PROGRAM MAIN
VAR
	iCounter 	: INT;
	
	bToggle		: BOOL;
	bReset		: BOOL;
	sText		: STRING; 
	
	stMyVar		: ST_MyType;
END_VAR


IF bToggle THEN
	sText := 'Stop';
	iCounter := (iCounter + 1) MOD 1000;
	IF iCounter = 0 THEN
		bToggle := FALSE;
	END_IF;	
ELSE
	sText := 'Start';
	IF bReset THEN
		bReset := FALSE;
		iCounter := 0;
	END_IF
END_IF

Alarming();
AlarmingEx();
AlarmExtension();

END_PROGRAM

(* stored: Version 1.1.0.1, ProductVersion 3.1.4024.12
   POU MAIN: Id {aefbc799-9f83-4d00-8ae0-e06bdca1ee13}, SpecialFunc None *)
